//Enumeration for Machineunits
TYPE E_UnitName :
(
	eMachine		:= 1,
	eUnit_Apron			:= 2,
	eUnit_BackGauge		:= 3,
	eUnit_Clamp			:= 4,
	eUnit_Slitter		:= 5
	
	
)DINT;
END_TYPE

(* stored: Version 1.1.0.1, ProductVersion 3.1.4024.12
   DUT E_UnitName: Id {8739632a-22aa-4382-9f71-9f3d2db45aad} *)
